//==================================================================================================
//						Beckhoff Automation Poland
//							21.05.2018
//				Program  odczytujący informacje o tasku pierwszym.
//
// 	v1.1 || TC v 3.1.4022.16 || - zgodnosc ze standardem
// 	v1.0 || TC v 3.1.4020.14 || - pierwsza wersja
//==================================================================================================
PROGRAM P_TaskInfo
VAR_INPUT
	bReset						: BOOL;
END_VAR
VAR_OUTPUT
	bOK							: BOOL;						// Brak bledow i ostrzezen
	bWarning					: BOOL;						// Ostrzezenie - nie wystepuja w tym podprogramie - wystepuja dla zachowania spojnosci
	bError						: BOOL;						// Zbiorcza flaga bledow
	udiErrorID					: UDINT;
	sErrorDescription			: WSTRING;
END_VAR
VAR
	fbTaskInfo					: FB_TaskInfo;
	rtError						: R_TRIG;
END_VAR

bError 							:= fbTaskInfo.bError; 		// Dla jednego tasku. W przypadku wiekszej ilosci taskow trzeba dopisac reszte.
bOk 							:= NOT bError;
fbTaskInfo.bReset				:= bReset;


fbTaskInfo();


rtError									(CLK:= bError);

IF rtError.Q THEN
	udiErrorID							:= 96;                                            
	sErrorDescription					:= "Błąd sterownika | Błąd programu sprawdzającego cykl sterownik";	
END_IF

IF NOT bError THEN
	udiErrorID							:= 0;	
	sErrorDescription					:= "";
END_IF

END_PROGRAM

(* stored: Version 1.1.0.1, ProductVersion 3.1.4026.13, FileIdentifier d87755bcaf70636e5fd05a3da1ebbd84d9870613, FileSignature 7193d3bae97d34a268a66880550af11ec3be8354310fd5077beef7068565f721622a42a5515470fcf787991c1e44189733239878a75c743e28a7ea6529127e6be6bbc1d37db1b825f653a2607505a169d0b7bb06448831e914de6f40c46e84d9069f2197063b34891984ab9dfa8da50b8969897ebeee21526536007f235ddbf4ad8fc255004709f721847262f3f08e3d006d5c3cc3ceb949ecd438a14fccddce8e7e46f76c529edd810708a149cdf1f6c296aaaf9f0e7799521649119e232d74fb7205f339922571c9c9a9af1e586d4019c9702b564fd69740265382c7f4f49d4d17b595e4eef0b2b3d8968c6ce617fab8c19dbd5eec73f99bbb1298149710f0
   POU P_TaskInfo: Id {963be1aa-f497-42e7-bc03-3e87922b27c9}, SpecialFunc None *)
